// TIA Portal V17 export
// export: Created 2023-02-13T11:05:56.575601Z, ExportSetting WithDefaults, DisplayName Totally Integrated Automation Portal, DisplayVersion V17, DisplayName TIA Portal Openness, DisplayVersion V17, DisplayName TIA Portal Teamcenter Gateway, DisplayVersion V17, DisplayName TIA Portal Version Control Interface, DisplayVersion V17, DisplayName SINAMICS Startdrive Advanced, DisplayVersion V17, DisplayName SINAMICS Startdrive G130, G150, S120, S150, SINAMICS MV, S210, DisplayVersion V17, DisplayName SINAMICS Startdrive G110M, G120, G120C, G120D, G120P, G115D, DisplayVersion V17, DisplayName STEP 7 Professional, DisplayVersion V17, DisplayName STEP 7 Safety, DisplayVersion V17, DisplayName WinCC Professional, DisplayVersion V17
VAR_GLOBAL   // PLC tag table "Timer"
   timerDrainTHE1_MS AT %MD30 : DInt;
   timerDrainTHE2_MS AT %MD34 : DInt;
   Timer_DrainSP AT %MD38 : DInt;
   timerDrainTHE1_ACT_MS AT %MD42 : DInt;
   timerDrainTHE2_ACT_MS AT %MD46 : DInt;
END_VAR
